(* IEC 61131-3 sources: RL_MAR/experiments/comparison/llm4plc/results/deepseek-ai-DeepSeek-V3.2_20260506_104945/20260506_105751, 3 files *)

(* ---- generated_code_iteration_0.st ---- *)
START_ST
FUNCTION_BLOCK RandomNumberGenerator
VAR_INPUT
    minValue : DINT;
    maxValue : DINT;
    randomSeed_in : DINT;
END_VAR
VAR_OUTPUT
    error : BOOL;
    status : WORD;
    randomNumber : DINT;
END_VAR
VAR
    state : INT;
    prevState : INT;
    internalSeed : DINT;
    range : DINT;
    tempRandom : DINT;
END_VAR

CASE state OF
    0: (* STATE 0: INITIALIZE / IDLE *)
        (* Outputs: error = FALSE (or previous value held), status = 16#0000 (or previous), randomNumber = 0 (or previous) *)
        (* No forced output changes here to hold previous values *)
        (* Transition: On every scan cycle when the function block is called, transition immediately to validation. *)
        state := 1;
        prevState := 0;

    1: (* STATE 1: VALIDATE RANGE *)
        IF minValue > maxValue THEN
            (* Range error: set outputs and return to idle *)
            error := TRUE;
            status := 16#8200;
            randomNumber := 0;
            state := 0;
        ELSE
            (* Range valid: set outputs and proceed to generation *)
            error := FALSE;
            status := 16#0000;
            state := 2;
        END_IF;
        prevState := 1;

    2: (* STATE 2: GENERATE RANDOM NUMBER *)
        (* Ensure seed is positive: use absolute value *)
        internalSeed := ABS(randomSeed_in);
        IF internalSeed = 0 THEN
            internalSeed := 1; (* Avoid zero seed to prevent modulo issues *)
        END_IF;

        (* Compute range for modulo operation *)
        range := maxValue - minValue + 1;
        IF range <= 0 THEN
            (* Should not happen as validated in state 1, but as safety fallback *)
            error := TRUE;
            status := 16#8200;
            randomNumber := 0;
        ELSE
            (* Generate random number using modulo arithmetic *)
            tempRandom := internalSeed MOD 32768; (* Simple pseudo-random step *)
            tempRandom := (tempRandom * 1103515245 + 12345) MOD 2147483648; (* Linear congruential generator for better distribution *)
            tempRandom := ABS(tempRandom);
            randomNumber := minValue + (tempRandom MOD range);

            (* Set outputs *)
            error := FALSE;
            status := 16#0000;
        END_IF;

        (* Return to idle *)
        state := 0;
        prevState := 2;

    ELSE
        (* Fallback: reset to state 0 *)
        state := 0;
END_CASE;
END_FUNCTION_BLOCK
END_ST

(* ---- generated_code_iteration_2.st ---- *)
START_REASON
The validation feedback indicates a type conversion error: "cannot convert type 'LINT' to type 'DINT'" in the CODESYS compiler. This error persists despite my previous attempt to fix it. Looking at the code, the issue likely occurs in state 2 where I used `DINT_TO_LINT` and `LINT_TO_DINT` conversions, but the compiler still complains about converting LINT to DINT. Specifically, the line `tempRandom := DINT_TO_LINT(internalSeed) * 16807;` attempts to assign a LINT value (result of multiplication) to a DINT variable `tempRandom`, causing the error. Even though I intended to use a temporary LINT, `tempRandom` is declared as DINT, so the assignment is invalid.

To resolve this, I need to avoid any implicit or explicit LINT to DINT conversions in assignments. Since the multiplication `internalSeed * 16807` can exceed DINT range (max 2,147,483,647), I must handle it without causing type mismatches. I can use a different algorithm that stays within DINT bounds or use explicit LINT variables for intermediate calculations and then safely convert to DINT using proper casting.

I'll modify the code as follows:
1. Declare a temporary LINT variable (e.g., `tempLint`) to hold the multiplication result.
2. Perform the calculation in LINT: `tempLint := DINT_TO_LINT(internalSeed) * 16807;`
3. Use `MOD` with a LINT modulus (2147483647, which is within LINT range) and store the result in `tempLint`.
4. Convert the LINT result back to DINT using `LINT_TO_DINT` and assign to a DINT variable.
5. Ensure all assignments are type-compatible.

Additionally, I'll simplify the algorithm to avoid unnecessary complexity and ensure the state machine works correctly. I'll also remove the `prevState` variable if not required, but I'll keep it for debugging if needed.

Let's implement these changes in the corrected code.
END_REASON

START_ST
FUNCTION_BLOCK RandomNumberGenerator
VAR_INPUT
    minValue : DINT;
    maxValue : DINT;
    randomSeed_in : DINT;
END_VAR
VAR_OUTPUT
    error : BOOL;
    status : WORD;
    randomNumber : DINT;
END_VAR
VAR
    state : INT;
    internalSeed : DINT;
    range : DINT;
    tempRandom : DINT;
    tempLint : LINT; // Temporary LINT variable for calculations
END_VAR

CASE state OF
    0: (* STATE 0: INITIALIZE / IDLE *)
        error := FALSE;
        status := 16#0000;
        randomNumber := 0;
        state := 1;

    1: (* STATE 1: VALIDATE RANGE *)
        IF minValue > maxValue THEN
            error := TRUE;
            status := 16#8200;
            randomNumber := 0;
            state := 0;
        ELSE
            error := FALSE;
            status := 16#0000;
            state := 2;
        END_IF;

    2: (* STATE 2: GENERATE RANDOM NUMBER *)
        internalSeed := ABS(randomSeed_in);
        IF internalSeed = 0 THEN
            internalSeed := 1;
        END_IF;

        range := maxValue - minValue + 1;
        IF range <= 0 THEN
            error := TRUE;
            status := 16#8200;
            randomNumber := 0;
        ELSE
            // Use LINT for intermediate calculation to avoid overflow
            tempLint := DINT_TO_LINT(internalSeed) * 16807;
            tempLint := tempLint MOD 2147483647; // Modulus operation in LINT
            tempRandom := LINT_TO_DINT(tempLint); // Convert back to DINT

            internalSeed := tempRandom; // Update seed (though not persistent)
            randomNumber := minValue + (tempRandom MOD range);

            error := FALSE;
            status := 16#0000;
        END_IF;

        state := 0;

    ELSE
        state := 0;
        error := TRUE;
        status := 16#8000;
        randomNumber := 0;
END_CASE;
END_FUNCTION_BLOCK
END_ST

(* ---- generated_code_iteration_1.st ---- *)
START_REASON
The validation feedback indicates a type conversion error: "cannot convert type 'LINT' to type 'DINT'". This error likely occurs in the calculation within state 2, where operations on DINT variables might produce intermediate results that exceed the DINT range (32-bit signed integer), causing the compiler to treat them as LINT (64-bit signed integer). Specifically, the line `tempRandom := (tempRandom * 1103515245 + 12345) MOD 2147483648;` involves multiplication of two DINT values (tempRandom and 1103515245), which can result in a value beyond the DINT range, leading to an implicit LINT conversion. The MOD operation with 2147483648 (which is 2^31, a LINT literal) then attempts to assign an LINT result back to a DINT variable (tempRandom), causing the type mismatch.

To fix this, I need to ensure all intermediate calculations stay within DINT range or explicitly handle type conversions. Since the requirement is to generate a random number within a DINT range, I can adjust the algorithm to use DINT-safe operations. One approach is to use a simpler pseudo-random generator that avoids large multiplications or to use built-in functions if available, but given the structured text constraints, I'll modify the calculation to prevent overflow. I can break down the multiplication or use a different constant. Alternatively, I can use type casting to LINT for the calculation and then cast back to DINT, but this might complicate things. Instead, I'll use a smaller multiplier or implement a shift-based method. However, for simplicity and to avoid LINT conversions, I'll replace the linear congruential generator with a simpler algorithm that uses DINT-friendly operations, such as a basic modulo generator with a seed update.

I'll revise state 2 to:
1. Use the internalSeed directly for generation.
2. Update the seed using a DINT-safe formula: e.g., `internalSeed := (internalSeed * 1103515245 + 12345) MOD 2147483647;` but this still risks LINT conversion. To avoid this, I can use `MOD` with a DINT-compatible modulus (e.g., 32767) or use bitwise operations. Since DINT in CODESYS is 32-bit, I'll use a modulus of 2147483647 (2^31 -1, which fits in DINT) and ensure multiplication doesn't overflow by using type casting to LINT temporarily, then convert back. But the feedback explicitly warns against LINT to DINT conversion, so I need a different approach.

I'll implement a simple pseudo-random algorithm using the `RAND` function if available, but since this is a function block without external functions, I'll use a basic algorithm: `internalSeed := (internalSeed * 1103515245 + 12345) MOD 2147483647;` and handle the multiplication by explicitly casting to LINT for the calculation, then cast back to DINT using truncation. However, CODESYS might still treat the literal 2147483647 as LINT if it's beyond DINT range? 2147483647 is within DINT range (max positive DINT is 2147483647), so it should be DINT. The issue is the multiplication result may exceed DINT, causing implicit LINT. To avoid this, I can use `MOD` after each step or use a smaller multiplier.

Given the constraints, I'll simplify: use `tempRandom := (internalSeed * 1103515245 + 12345) MOD 2147483647;` and ensure all operands are DINT, but the product may exceed, so I'll use a LINT temporary variable, then convert to DINT. But the error is about converting LINT to DINT, so I need to explicitly handle the conversion. I can declare a temporary LINT variable, perform the calculation in LINT, then assign to DINT using type conversion. However, CODESYS may require explicit casting functions like `DINT_TO_LINT` and `LINT_TO_DINT`. To keep it simple, I'll change the algorithm to use a smaller multiplier that doesn't cause overflow, e.g., 16807 (a common multiplier for pseudo-random generators). This should keep results within DINT range when using modulus 2147483647.

Revised plan for state 2:
- Use multiplier 16807 and modulus 2147483647.
- Calculate: `tempRandom := (internalSeed * 16807) MOD 2147483647;`
- Then add 12345 and mod again if needed, but to avoid complexity, I'll use a standard linear congruential generator with these constants.
- Update internalSeed for next call, but since internalSeed is not persistent across calls (it's reinitialized each time), I'll just compute tempRandom directly.

Also, ensure range calculation is correct and all outputs are set properly. I'll also initialize variables in state 0 to default values to avoid holding previous values incorrectly.

Finally, I'll structure the code with proper state transitions and output settings.
END_REASON

START_ST
FUNCTION_BLOCK RandomNumberGenerator
VAR_INPUT
    minValue : DINT;
    maxValue : DINT;
    randomSeed_in : DINT;
END_VAR
VAR_OUTPUT
    error : BOOL;
    status : WORD;
    randomNumber : DINT;
END_VAR
VAR
    state : INT;
    prevState : INT;
    internalSeed : DINT;
    range : DINT;
    tempRandom : DINT;
END_VAR

CASE state OF
    0: (* STATE 0: INITIALIZE / IDLE *)
        (* Initialize outputs to default values *)
        error := FALSE;
        status := 16#0000;
        randomNumber := 0;
        (* Transition to validation on next scan *)
        state := 1;
        prevState := 0;

    1: (* STATE 1: VALIDATE RANGE *)
        IF minValue > maxValue THEN
            (* Range error: set outputs and return to idle *)
            error := TRUE;
            status := 16#8200;
            randomNumber := 0;
            state := 0;
        ELSE
            (* Range valid: proceed to generation *)
            error := FALSE;
            status := 16#0000;
            state := 2;
        END_IF;
        prevState := 1;

    2: (* STATE 2: GENERATE RANDOM NUMBER *)
        (* Ensure seed is positive and non-zero *)
        internalSeed := ABS(randomSeed_in);
        IF internalSeed = 0 THEN
            internalSeed := 1;
        END_IF;

        (* Compute range for modulo operation *)
        range := maxValue - minValue + 1;
        IF range <= 0 THEN
            (* Fallback error, though validated in state 1 *)
            error := TRUE;
            status := 16#8200;
            randomNumber := 0;
        ELSE
            (* Generate pseudo-random number using a DINT-safe linear congruential generator *)
            (* Constants: multiplier a = 16807, modulus m = 2147483647 (2^31 - 1) *)
            (* Formula: internalSeed = (internalSeed * 16807) MOD 2147483647 *)
            (* Use temporary LINT for multiplication to avoid overflow, then convert back to DINT *)
            tempRandom := DINT_TO_LINT(internalSeed) * 16807;
            tempRandom := LINT_TO_DINT(tempRandom MOD 2147483647);

            (* Update internalSeed for potential future use, though not stored persistently *)
            internalSeed := tempRandom;

            (* Scale to desired range *)
            randomNumber := minValue + (tempRandom MOD range);

            (* Set outputs *)
            error := FALSE;
            status := 16#0000;
        END_IF;

        (* Return to idle *)
        state := 0;
        prevState := 2;

    ELSE
        (* Fallback: reset to state 0 *)
        state := 0;
        error := TRUE;
        status := 16#8000;
        randomNumber := 0;
END_CASE;
END_FUNCTION_BLOCK
END_ST
